Staubli VAL3: insert_aIn.pgx

public program insert_aIn(string x_sItem (dimensions=1), bool x_bActive (dimensions=1), aio x_aDio (dimensions=1))
begin
  // insert a new IO
  if isDefined(aInput[x_sItem])==false and ioStatus(x_aDio)>=0
    insert(aInput[x_sItem])
    aInput[x_sItem].bActive=x_bActive
    aInput[x_sItem].sID=x_sItem
    aInput[x_sItem].sName=x_sItem
    aioLink(aInput[x_sItem].aAio,x_aDio)
    aInput[x_sItem].bEnable=true
  endIf
end
